// Mitsubishi GX Works2 project: tes-modbus   PLC: FX3U/FX3UC

PROGRAM MAIN
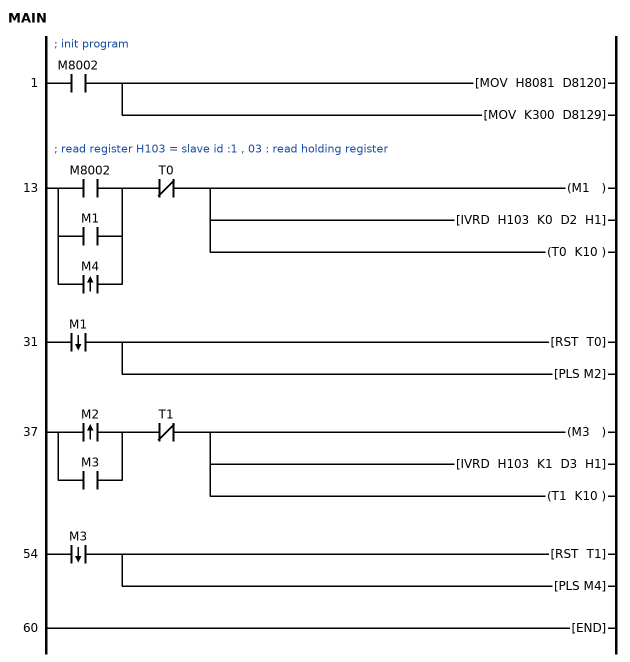
; init program
1     LD      M8002
      MOV     H8081 D8120
      MOV     K300 D8129
; read register H103 = slave id :1 , 03 : read holding register
13    LD      M8002
      OR      M1
      ORP     M4
      ANI     T0
      OUT     M1
      IVRD    H103 K0 D2 H1
      OUT     T0 K10
31    LDF     M1
      RST     T0
      PLS     M2
37    LDP     M2
      OR      M3
      ANI     T1
      OUT     M3
      IVRD    H103 K1 D3 H1
      OUT     T1 K10
54    LDF     M3
      RST     T1
      PLS     M4
60    END
END_PROGRAM
